(* IEC 61131-3 sources: Mizera_Tube/Plc (part 14) *)

(* ---- RES_IPG.plc ---- *)
*******************************************************************************
*   RES_IPG.PLC
*   ESAutomotion
*   LASER machine
*******************************************************************************
VAR
#include "Cnc.inc"
#include "RemContr.inc"
END_VAR

VAR_IN_OUT
#include "mem.inc"
END_VAR

#include "Iol.inc"
#include "res_ipg.inc"

*******************************************************************************
*   RESONATOR: IPG (YLR / YLS type)
*******************************************************************************
FUNCTION_BLOCK IPG
VAR_INPUT
xSIM:       BOOL;           * Laser in simulation (become from LSR_GEST)
xType:      DWORD;          * 0=YLS, 1=YLR
xReset:     BOOL;           * reset
xEmer:      BOOL;           * emerg
xEmission:  BOOL;           * Emission command
END_VAR

VAR_OUTPUT
yError:     DWORD;          * error
yWarning:   DWORD;          * warning
yState:     BOOL;           * 1=EMISSION ON, 0=EMISSION OFF
END_VAR

VAR
Appoggio:               BOOL;
YLSseries:              BOOL;
YLRseries:              BOOL;
AutoSwitchOn:           BOOL;
Aux_Allarme:            BOOL;
Feedback_Emission_ON:   BOOL;
TON_LASER_REQ:          TON;        * autostart: Laser request OUT
TON_LASER_SWITCH:       TON;        * autostart: Laser switch on OUT
TON_ANALOG_CONTROL:     TON;        * autostart: analog control OUT
TON1:                   TON;        * timeout 1
TON2:                   TON;        * timeout 1
TON3:                   TON;        * timeout 1
RTRIG_RESET:            R_TRIG;     * trigger on reset button
Guide_Las:              BOOL;
CTU_PULS_Guide_Las:     CTU;
RTRIG_REM_GUIDE_LAS:    R_TRIG;
R_TRIG_RemLaserOn:      R_TRIG;
END_VAR

*******************************************************************************
LD   ALWAYS_ZERO                   ** PLCFLAGS.0  Flag sempre stato off
ST   YLSseries
LD   ALWAYS_ONE                    ** PLCFLAGS.1  Flag sempre stato on
ST   YLRseries

LD   xType                         ** 0=YLS, 1=YLR
EQ   0
JMPCN IsYLR

LD   ALWAYS_ONE                    ** PLCFLAGS.1  Flag sempre stato on
ST   YLSseries
LD   ALWAYS_ZERO                   ** PLCFLAGS.0  Flag sempre stato off
ST   YLRseries

IsYLR:

LD   %Par0.0
ANDN (
LD   xReset                        ** reset
ANDN  I_B8_POWER_SUPPLY            ** IPG power supply status
)
ANDN xEmer                         ** emerg
ST   AutoSwitchOn

CAL  TON_LASER_REQ(IN=AutoSwitchOn, PT=0) ** autostart: Laser request OUT

LD   AutoSwitchOn
AND  O_A1_LASER_REQ                ** IPG Richiesta Laser
ST   Appoggio

CAL  TON_LASER_SWITCH(IN=Appoggio, PT=1000) ** autostart: Laser switch on OUT

LD   AutoSwitchOn
AND  O_C1_LASER_SWITCH             ** IPG Laser Switch ON
ST   Appoggio

CAL  TON_ANALOG_CONTROL(IN=Appoggio, PT=1000) ** autostart: analog control OUT

CAL  RTRIG_RESET(CLK=xReset)       ** trigger on reset button

LD   RTRIG_RESET.Q
JMPCN NoReset

LD   0
ST   yError                        ** error
ST   yWarning                      ** warning

LD   ALWAYS_ZERO                   ** PLCFLAGS.0  Flag sempre stato off
ST   yState                        ** 1=EMISSION ON, 0=EMISSION OFF

NoReset:

*******************************************************************************
*   A01 Laser request (wait Laser_ASSIGNED)
*******************************************************************************
CAL  R_TRIG_RemLaserOn(CLK=RemContrLaserOn)
LD   R_TRIG_RemLaserOn.Q
AND  O_A1_LASER_REQ
R    BTN_LASER_REQUEST

LD   R_TRIG_RemLaserOn.Q
ANDN O_A1_LASER_REQ
S    BTN_LASER_REQUEST

LD   BTN_LASER_REQUEST
ANDN AutoSwitchOn
AND  YLSseries
OR (
LD   BTN_LASER_REQUEST
ANDN AutoSwitchOn
AND  YLRseries
AND  I_B8_POWER_SUPPLY             ** IPG power supply status (IW1.6)
)
OR   TON_LASER_REQ.Q
ANDN xSIM                          ** Laser in simulation (become from LSR_GEST)
ST   O_A1_LASER_REQ                ** IPG Richiesta Laser (QW3.11)

*******************************************************************************
*   C01 POWER SUPPLY ON (wait B8 power supply status)
*******************************************************************************
LD   BTN_POWER_ON
ANDN AutoSwitchOn
OR   TON_LASER_SWITCH.Q
AND  O_A1_LASER_REQ                ** IPG Richiesta Laser
AND  I_B7_LASER_ASSIGNED           ** IPG Laser ASSIGNED
ANDN xSIM                          ** Laser in simulation (become from LSR_GEST)
AND  YLSseries
ST   O_C1_LASER_SWITCH             ** IPG Laser Switch ON

*******************************************************************************
*   A05 Guide laser ON
*******************************************************************************
CAL  RTRIG_REM_GUIDE_LAS(CLK:=RemContrGuideLas)        * Xhc_Puls.17 Laser shut

CAL  CTU_PULS_Guide_Las(CU:=RTRIG_REM_GUIDE_LAS.Q,R=CTU_PULS_Guide_Las.Q,PV=2)

LD   CTU_PULS_Guide_Las.CV
EQ   1
ST   Guide_Las

LD   BTN_GUIDE_ON
OR   Guide_Las
ANDN xSIM                          ** Laser in simulation (become from LSR_GEST)
ST   O_A5_GUIDE_LASER              ** IPG Laser spot guide ON

*******************************************************************************
*   A06 Analog control ON
*******************************************************************************
LD   BTN_ANALOG_ON
OR   TON_ANALOG_CONTROL.Q
ANDN xSIM                          ** Laser in simulation (become from LSR_GEST)
ST   O_A6_ANALOG_CONTROL           ** IPG Controllo analogico ON

*******************************************************************************
*   A03 Enable internal control
*******************************************************************************
LD   BTN_INT_ON
ANDN xSIM                          ** Laser in simulation (become from LSR_GEST)
ST   O_A3_INT_CONTROL              ** IPG Abilitazione Controllo interno

*******************************************************************************
*   A04 Reset
*******************************************************************************
LD   BTN_RESET
*OR   xReset                        ** reset
ANDN xSIM                          ** Laser in simulation (become from LSR_GEST)
ST   O_A4_LASER_RESET              ** IPG Resetta errori

*******************************************************************************
*   START PROGRAM
*******************************************************************************
*LD   xEmission                     ** Emission command
*ANDN xSIM                          ** Laser in simulation (become from LSR_GEST)
*ST   O_A2_LASER_PROG_RUN           ** IPG (START PROGRAM)

*******************************************************************************
*   ERROR
*******************************************************************************
*** Allarme errore laser (B4)
LD   I_B4_LASER_ERROR              ** IPG YLS YLR Laser in Alarm status
ST   yError.0

*** Allarme laser non attivo (A2 senza B1)
LD   O_A2_LASER_PROG_RUN           ** IPG (START PROGRAM)
ANDN I_B1_LASER_READY              ** IPG Laser internal main power supply ON (Aux Power ON)
ST   yError.1

*** Allarme laser non assegnato (A1 senza B7)
LD   O_A1_LASER_REQ                ** IPG Richiesta Laser
ANDN I_B7_LASER_ASSIGNED           ** IPG Laser ASSIGNED
ST    Aux_Allarme

CAL  TON1(IN=Aux_Allarme,PT=3000)  ** timeout 1
LD   TON1.Q
ST   yError.2

*** Allarme laser non attivo (C1 senza B8)
LD   O_C1_LASER_SWITCH             ** IPG Laser Switch ON
ANDN I_B8_POWER_SUPPLY             ** IPG power supply status
ST   Aux_Allarme

CAL  TON2(IN=Aux_Allarme,PT=5000)  ** timeout 1
LD   TON2.Q
ST   yError.3

*** Allarme Trascorso tempo massimo attesa segnale emission on dal laser
LD   O_A2_LASER_PROG_RUN           ** IPG (START PROGRAM)
ANDN I_B2_EMISSION_ON              ** IPG Emission ON
ST   Feedback_Emission_ON

CAL  TON3(IN=Feedback_Emission_ON,PT=3000) ** timeout 1

LD   TON3.Q
ST   yError.4

*******************************************************************************
*   WARNING
*******************************************************************************
*** Messaggio laser in stato di pre-allarme (B13)

LD   I_B13_AVVERTENZA              ** IPG WARNING OUT
ST   yWarning.0

LD   O_A2_LASER_PROG_RUN           ** IPG (START PROGRAM)
***AND  I_B2_EMISSION_ON              ** IPG Emission ON
ST   yState                        ** 1=EMISSION ON, 0=EMISSION OFF

*******************************************************************************
*   HMI
*******************************************************************************

*** Buttons

LD   O_A1_LASER_REQ                ** IPG Richiesta Laser
ST   %Leds0.0
LD   O_C1_LASER_SWITCH             ** IPG Laser Switch ON
ST   %Leds0.1
LD   O_A4_LASER_RESET              ** IPG Resetta errori
ST   %Leds0.2
LD   O_A3_INT_CONTROL              ** IPG Abilitazione Controllo interno
ST   %Leds0.3
LD   O_A6_ANALOG_CONTROL           ** IPG Controllo analogico ON
ST   %Leds0.4
LD   O_A5_GUIDE_LASER              ** IPG Laser spot guide ON
ST   %Leds0.5
LD   O_A2_LASER_PROG_RUN           ** IPG (START PROGRAM)
ST   %Leds0.6

*** Feedback

LD   I_B7_LASER_ASSIGNED           ** IPG Laser ASSIGNED
ST   %Leds1.0
LD   I_B8_POWER_SUPPLY             ** IPG power supply status
ST   %Leds1.1
LD   I_B3_INT_CONTROL              ** IPG Controllo interno abilitato
ST   %Leds1.2
LD   I_B6_ANALOG_CONTROL           ** IPG Controllo analogico ON
ST   %Leds1.3
LD   I_B5_LASER_GUIDE              ** IPG Laser guida ON
ST   %Leds1.4
LD   I_B1_LASER_READY              ** IPG Laser internal main power supply ON (Aux Power ON)
ST   %Leds1.5
LD   I_B2_EMISSION_ON              ** IPG Emission ON
ST   %Leds1.6
LD   I_B13_AVVERTENZA              ** IPG WARNING OUT
ST   %Leds1.7
LD   I_B4_LASER_ERROR              ** IPG YLS YLR Laser in Alarm status
ST   %Leds1.8

*** If laser in simulation

LD   xSIM                          ** Laser in simulation (become from LSR_GEST)
JMPCN NoLaserInSIM
LD   0
ST   yError                        ** error
ST   yWarning                      ** warning

LD   xEmission                     ** Emission command
ST   yState                        ** 1=EMISSION ON, 0=EMISSION OFF
NoLaserInSIM:

END_FUNCTION_BLOCK

(* ---- RestFB.plc ---- *)
**************************************************
* New state machine to restart the machine after
* an hold command or tip touch event
**************************************************

FUNCTION_BLOCK Restart_Cut

VAR
State:              DWORD;
ActualAttempts:     DWORD;
PrevCountAttempt:   DWORD;
RetraceTimeout:     DWORD;

ResetCounter:       BOOL;
MaxAttemptsDone:    BOOL;

TON_RETR_DONE:      TON;
TON_RESCOUNT:       TON;
FTRIG_END_RETRACE:  F_TRIG;

END_VAR

VAR_INPUT
xProg_Run:      BOOL;
xTip_Touch:     BOOL;
xZupExecuted:   BOOL;
xMachineInHold: BOOL;
xRetraceOn:     BOOL;
xAttempts:      DWORD;
END_VAR

VAR_OUTPUT
yZupRequest:    BOOL;
yStartRetrace:  BOOL;
yStartProg:     BOOL;
yHoldProg:      BOOL;
yInibTipTouch:  BOOL;
END_VAR

*********************************************************************

LD   3000
ST   RetraceTimeout

LDN  xProg_Run
JMPCN no_ResetVar

LD   0
ST   yZupRequest
ST   yStartRetrace
ST   yStartProg
ST   yHoldProg
ST   yInibTipTouch
ST   State

LD   1
ST   ActualAttempts
ST   PrevCountAttempt
no_ResetVar:

*****************************
* Attempt counter

LD   ActualAttempts
GT   xAttempts
ST   MaxAttemptsDone

LD   ActualAttempts
EQ   PrevCountAttempt
ANDN MaxAttemptsDone
ST   ResetCounter

CAL  TON_RESCOUNT (IN:=ResetCounter,PT:=20000)

LD   TON_RESCOUNT.Q
JMPCN no_res_count
LD   0
ST   PrevCountAttempt
ST   ActualAttempts
no_res_count:
******************************

*********************************************************************
*   STATO=0
*   In case of tip touch this state makes a request to the regulator
*   to bring up the head
*********************************************************************
LD   State
EQ   0
JMPCN STATE0_end

R    yStartProg

LD   ActualAttempts
ST   PrevCountAttempt

LD   xTip_Touch
AND  xProg_Run
ANDN MaxAttemptsDone
JMPCN STATE0_endif_A

** assume stay here just one scan
LD  ActualAttempts
ADD 1
ST  ActualAttempts
**

S   yZupRequest
S   yInibTipTouch

LD  10
ST  State

STATE0_endif_A:
JMP state_machine_end

STATE0_end:

CAL  TON_RETR_DONE (IN:=yStartRetrace,PT:=RetraceTimeout)
CAL  FTRIG_END_RETRACE(CLK=xRetraceOn)

*********************************************************************
*   STATO=10
*   Wait that the machine is in hold then send the request of retrace back
*********************************************************************
LD   State
EQ   10
JMPCN STATE10_end

LD   xZupExecuted
AND  xMachineInHold
JMPCN STATE10_endif_A

S  yStartRetrace

LD  11
ST  State

STATE10_endif_A:
JMP state_machine_end

STATE10_end:

*********************************************************************
*   STATO=11
*   Wait that the machine is in hold then send the request of retrace back
*********************************************************************
LD   State
EQ   11
JMPCN STATE11_end

LD   FTRIG_END_RETRACE.Q
OR (
LD   TON_RETR_DONE.Q
ANDN xRetraceOn
)
JMPCN no_retrace_end

R   yStartRetrace
R   yInibTipTouch
R   yZupRequest
S   yStartProg

LD  0
ST  State

no_retrace_end:
JMP state_machine_end

STATE11_end:

*********************************************************************
state_machine_end:

END_FUNCTION_BLOCK

(* ---- RToolSur.plc ---- *)
*=========================================================================
* VRTC GATEWAY VARIABLES SECTION
*=========================================================================
#funcdec "ASSI.plc"
#funcdec "CNC.plc"
#funcdec "StatMReg.plc"

VAR
REG_MAC:  REG_STATE_MACHINE;
vrtcExTool:         VRTC_EX;
vrtcExSurface:      VRTC_EX;

plcVrtcHandling:       BOOL;
firstCallToPlcHandler:  BOOL;

toolCommandToggle:      BOOL;
surfaceCommandToggle:   BOOL;
appoggio:               BOOL;

TR_ToolVrtcToggle:      TRIG;
TR_SurfaceVrtcToggle:   TRIG;
RTR_PlcVrtcHandling:    R_TRIG;
cosAngle:               DWORD;
ActVPBSelect:           DWORD;
TP_reset:               TP;

SensorGain:             DWORD;

END_VAR

VAR_IN_OUT
UVH_COMMAND_0                          AT %uvhCommand0;
UVH_COMMAND_MACHINE_MODE               AT %uvhCommand1;
UVH_COMMAND_PLC_VRTC_HANDLING          AT %uvhCommand0.1;
UVH_COMMAND_START_COMMAND              AT %uvhCommand0.2;
UVH_COMMAND_FREEZE_REGOL               AT %uvhCommand0.3;
UVH_COMMAND_JUMP                       AT %uvhCommand0.4;
UVH_COMMAND_L10                        AT %uvhCommand0.5;
UVH_COMMAND_L3                         AT %uvhCommand0.6;
UVH_STATUS_PLC_VRTC_HANDLING           AT %uvhStatus0.1;
UVH_STATUS_MACHINE_MODE                AT %uvhStatus1;
UVH_STATUS_COMMAND_RUNNING             AT %uvhStatus0.2;

UVH_TOOL_COMMAND_RESET                 AT %uvhToolCommand0.0;
UVH_TOOL_COMMAND_SIMUL                 AT %uvhToolCommand0.1;
UVH_TOOL_COMMAND_MOVE_TO_TARGET        AT %uvhToolCommand0.2;
UVH_TOOL_COMMAND_RES_POS_INT           AT %uvhToolCommand0.3;
UVH_TOOL_COMMAND_POS_LIM_DISAB         AT %uvhToolCommand0.4;
UVH_TOOL_COMMAND_DE_OVERLAP_ENAB       AT %uvhToolCommand0.5;
UVH_TOOL_COMMAND_ERROR_AMP_ENAB        AT %uvhToolCommand0.6;
UVH_TOOL_COMMAND_TOGGLE                AT %uvhToolCommand0.31;
UVH_TOOL_COMMAND_SIM_OFFSET_SET        AT %uvhToolCommand1;
UVH_TOOL_COMMAND_SETPOINT              AT %uvhToolCommand2;
UVH_TOOL_COMMAND_VECTOR_SELECT         AT %uvhToolCommand3;

UVH_TOOL_STATUS_SIGNAL_LOCK            AT %uvhToolStatus0.2;
UVH_TOOL_STATUS_TOGGLE_ACK             AT %uvhToolStatus0.31;
UVH_TOOL_STATUS_SIM_OFFSET_CUR         AT %uvhToolStatus1;
UVH_TOOL_STATUS_FLT_Q                  AT %uvhToolStatus2;

UVH_SURFACE_COMMAND_RESET              AT %uvhSurfaceCommand0.0;
UVH_SURFACE_COMMAND_SIMUL              AT %uvhSurfaceCommand0.1;
UVH_SURFACE_COMMAND_MOVE_TO_TARGET     AT %uvhSurfaceCommand0.2;
UVH_SURFACE_COMMAND_RES_POS_INT        AT %uvhSurfaceCommand0.3;
UVH_SURFACE_COMMAND_POS_LIM_DISAB      AT %uvhSurfaceCommand0.4;
UVH_SURFACE_COMMAND_DE_OVERLAP_ENAB    AT %uvhSurfaceCommand0.5;
UVH_SURFACE_COMMAND_ERROR_AMP_ENAB     AT %uvhSurfaceCommand0.6;
UVH_SURFACE_COMMAND_TOGGLE             AT %uvhSurfaceCommand0.31;
UVH_SURFACE_COMMAND_SIM_OFFSET_SET     AT %uvhSurfaceCommand1;
UVH_SURFACE_COMMAND_SETPOINT           AT %uvhSurfaceCommand2;
UVH_SURFACE_COMMAND_VECTOR_SELECT      AT %uvhSurfaceCommand3;

UVH_SURFACE_STATUS_SIGNAL_LOCK         AT %uvhSurfaceStatus0.2;
UVH_SURFACE_STATUS_TOGGLE_ACK          AT %uvhSurfaceStatus0.31;
UVH_SURFACE_STATUS_SIM_OFFSET_CUR      AT %uvhSurfaceStatus1;
UVH_SURFACE_STATUS_FLT_Q               AT %uvhSurfaceStatus2;

VRMON_Q_FLT_Q                          AT %VrMon_Q_Flt_Q;
VrSensorGain                          AT %VrSensorGain;
END_VAR

FUNCTION_BLOCK REG_T_S

VAR_INPUT

* Tool VRTC Input

xToolVrtcSetPoint:       DWORD;
xToolVrtcId:            DWORD;
xToolSim:                BOOL;

xLimDownSpeed:            BOOL;

xSensorRes:              DWORD;         * Capacitive sensor resolution (4095,32767,65535)
xNextPos_X_Jump_VRTC:    DWORD;         * X setpoint coordinate for jump
xNextPos_Y_Jump_VRTC:    DWORD;         * Y setpoint coordinate for jump
xNextPos_C_Jump_VRTC:    DWORD;         * C setpoint coordinate for jump
xNextPos_Z_Jump_VRTC:    DWORD;         * Z setpoint coordinate for jump

xInit_X_Posit_VRTC:      DWORD;         * X init jump position
xInit_Y_Posit_VRTC:      DWORD;         * Y init jump position
xInit_C_Posit_VRTC:      DWORD;         * C init jump position
xInit_Z_Posit_VRTC:      DWORD;         * C init jump position

xNextSetpVRTC:           DWORD;         * Setpoint after jump
xPrevSetpVRTC:           DWORD;         * last setpoint before jump
xDistEnabRegulVRTC:      DWORD;         * Distance from target to enab regulation during jump
xZDistStopProbeJVRTC:    DWORD;         * distance along Z to disable the probe vpbselector during jump

xActual_X_Posit_VRTC:    DWORD;         * X Actual position
xActual_Y_Posit_VRTC:    DWORD;         * Y Actual position
xActual_C_Posit_VRTC:    DWORD;         * C Actual position
xActual_Z_Posit_VRTC:    DWORD;         * Z Actual position

* Surface VRTC Input

xSurfVrtcId:            DWORD;
xSurfaceSim:            BOOL;
xLimSpeedPierc:           BOOL;
xAngleBev:              DWORD;
xSpeedForPiercing:        DWORD;                 * Speed for Z axi during piercing

xHead:                  DWORD;
xChannel:               DWORD;
xZtcp:                  DWORD;
xProbThreshold:         DWORD;
xSensorRange:           DWORD;
xFirstFirCost_VRTC:     DWORD;         * ms
xSecondFirCost_VRTC:    DWORD;         * ms
xDelayCost_VRTC:        DWORD;         * ms
xMove_Z_SetP_VRTC:        DWORD;

xMove_Z_VRTC:           BOOL;
xHold_VRTC:             BOOL;
xRealTimeFreeze:         BOOL;

END_VAR

VAR_OUTPUT
yWaitVRTC:               BOOL;
yIncSetPReachedVRTC:     BOOL;
yL3SetpointReachedVRTC:   BOOL;
END_VAR
*=========================================================================
* VRTC GATEWAY SECTION
*=========================================================================
***
* Vrtc Sensor gain settings

LD   xSensorRes
MUL  10000
DIV  xSensorRange
MUL  100
ST   SensorGain

PATH    %vrtc[xToolVrtcId]
LD   SensorGain
ST   VrSensorGain

PATH    %vrtc[xSurfVrtcId]
LD   SensorGain
ST   VrSensorGain

**

*** COMMON ***

LDN     %rc8.21                     * M_IDLE
JMPC    skip_vrtc_idle

    LD      0
    ST      UVH_COMMAND_0

skip_vrtc_idle:

LD      UVH_COMMAND_PLC_VRTC_HANDLING
ST      plcVrtcHandling

*** TOOL VRTC ***

* in cima
LD      UVH_TOOL_COMMAND_TOGGLE
ST      toolCommandToggle

CAL     TR_ToolVrtcToggle(CLK=toolCommandToggle)
LDN     TR_ToolVrtcToggle.Q
JMPC    skip_tool_vrtc_uvh_control

LD      UVH_TOOL_COMMAND_VECTOR_SELECT
ST      vrtcExTool.xVectorSelect

LD      UVH_TOOL_COMMAND_RESET
ST      vrtcExTool.xReset

LD      UVH_TOOL_COMMAND_SIMUL
ST      vrtcExTool.xSimul

LD      UVH_TOOL_COMMAND_MOVE_TO_TARGET
ST      vrtcExTool.xMoveToTarget

LD      UVH_TOOL_COMMAND_RES_POS_INT
ST      vrtcExTool.xResPosInt

LD      UVH_TOOL_COMMAND_POS_LIM_DISAB
ST      vrtcExTool.xPosLimDisab

LD      UVH_TOOL_COMMAND_DE_OVERLAP_ENAB
ST      vrtcExTool.xDeOverlapEnab

LD      UVH_TOOL_COMMAND_ERROR_AMP_ENAB
ST      vrtcExTool.xErrorAmpEnab

LD      UVH_TOOL_COMMAND_SIM_OFFSET_SET
ST      vrtcExTool.xSimOffsetSet

LD      UVH_TOOL_COMMAND_SETPOINT
ST      vrtcExTool.xSetPoint

skip_tool_vrtc_uvh_control:

*** SURFACE VRTC ***

* in cima
LD      UVH_SURFACE_COMMAND_TOGGLE
ST      surfaceCommandToggle

CAL     TR_SurfaceVrtcToggle(CLK=surfaceCommandToggle)
LDN     TR_SurfaceVrtcToggle.Q
JMPC    skip_surface_vrtc_uvh_control

LD      UVH_SURFACE_COMMAND_VECTOR_SELECT
ST      vrtcExSurface.xVectorSelect

LD      UVH_SURFACE_COMMAND_RESET
ST      vrtcExSurface.xReset

LD      UVH_SURFACE_COMMAND_SIMUL
ST      vrtcExSurface.xSimul

LD      UVH_SURFACE_COMMAND_MOVE_TO_TARGET
ST      vrtcExSurface.xMoveToTarget

LD      UVH_SURFACE_COMMAND_RES_POS_INT
ST      vrtcExSurface.xResPosInt

LD      UVH_SURFACE_COMMAND_POS_LIM_DISAB
ST      vrtcExSurface.xPosLimDisab

LD      UVH_SURFACE_COMMAND_DE_OVERLAP_ENAB
ST      vrtcExSurface.xDeOverlapEnab

LD      UVH_SURFACE_COMMAND_ERROR_AMP_ENAB
ST      vrtcExSurface.xErrorAmpEnab

LD      UVH_SURFACE_COMMAND_SIM_OFFSET_SET
ST      vrtcExSurface.xSimOffsetSet

LD      UVH_SURFACE_COMMAND_SETPOINT
ST      vrtcExSurface.xSetPoint

skip_surface_vrtc_uvh_control:

LDN     plcVrtcHandling
JMPCN   reset_vbselect

LD      0
ST      %vpbSelectors0

reset_vbselect:

*** COMMON ***

CAL     RTR_PlcVrtcHandling(CLK=plcVrtcHandling)
LD      RTR_PlcVrtcHandling.Q
ST      firstCallToPlcHandler

LDN     plcVrtcHandling
JMPC    skip_plc_handling
*XXX DO YOUR OWN PLC HANDLING cambio setpoint etc

 LD      xAngleBev                   * Bevel angle ofthe head
 COS
 ST      cosAngle

* State Machine FB

 LD      vrtcExSurface.xSimul
 ST      REG_MAC.xISO_S_SimEnab

 LD      vrtcExSurface.xErrorAmpEnab
 ST      REG_MAC.xISO_S_ErrAmp

 LD      vrtcExTool.xSimul
 ST      REG_MAC.xISO_T_SimEnab

 LD      vrtcExTool.xSetPoint
 ST      REG_MAC.xISO_T_SetPoint

 LD      vrtcExTool.xErrorAmpEnab
 ST      REG_MAC.xISO_T_ErrAmp

 LD      xFirstFirCost_VRTC
 ST      REG_MAC.xFirstFirCost         * ms

 LD      xSecondFirCost_VRTC
 ST      REG_MAC.xSecondFirCost        * ms

 LD      xDelayCost_VRTC
 ST      REG_MAC.xDelayCost         * ms

 LD      firstCallToPlcHandler
 ST      REG_MAC.xFirstPlcHandling

 LD      xProbThreshold
 ST      REG_MAC.xProbThres

 LD      xZtcp
 ST      REG_MAC.xZ_TCP

 LD      UVH_COMMAND_MACHINE_MODE
 ST      REG_MAC.xIsoPhase

 LD      vrtcExTool.yBusy
 ST      REG_MAC.xToolBusy

 LD      vrtcExSurface.yBusy
 ST      REG_MAC.xSurfaceBusy

 LD      vrtcExTool.ySignalLock
 ST      REG_MAC.xToolSignalLock

 LD      vrtcExSurface.ySignalLock
 ST      REG_MAC.xSurfSignalLock

 LD      xToolVrtcSetPoint         * [um]
 DIV     10
 ST      REG_MAC.xSetpoint

 LD      UVH_COMMAND_START_COMMAND
 ST      REG_MAC.xStartEx

 LD      xSensorRange
 ST      REG_MAC.xSensorRange

 LD      UVH_COMMAND_FREEZE_REGOL
 OR      xRealTimeFreeze
 ST      REG_MAC.xFreezeRegol

 LD      xNextPos_Y_Jump_VRTC          * Y setpoint coordinate for jump
 ST      REG_MAC.xNextPos_Y_Jump

 LD      xNextPos_X_Jump_VRTC          * X setpoint coordinate for jump
 ST      REG_MAC.xNextPos_X_Jump

 LD      xNextPos_C_Jump_VRTC          * C setpoint coordinate for jump
 ST      REG_MAC.xNextPos_C_Jump

 LD      xNextPos_Z_Jump_VRTC          * Z setpoint coordinate for jump
 ST      REG_MAC.xNextPos_Z_Jump

 LD      xInit_Y_Posit_VRTC            * Y init jump position
 ST      REG_MAC.xInit_Y_Posit

 LD      xInit_X_Posit_VRTC            * X init jump position
 ST      REG_MAC.xInit_X_Posit

 LD      xInit_C_Posit_VRTC            * C init jump position
 ST      REG_MAC.xInit_C_Posit

 LD      xInit_Z_Posit_VRTC            * Z init jump position
 ST      REG_MAC.xInit_Z_Posit

 LD      xActual_X_Posit_VRTC          * X Actual position
 ST      REG_MAC.xActual_X_Posit

 LD      xActual_C_Posit_VRTC          * C Actual position
 ST      REG_MAC.xActual_C_Posit

 LD      xActual_Z_Posit_VRTC          * C Actual position
 ST      REG_MAC.xActual_Z_Posit

 LD      xActual_Y_Posit_VRTC          * Y Actual position
 ST      REG_MAC.xActual_Y_Posit

 LD      UVH_COMMAND_JUMP
 ST      REG_MAC.xJumpReq

 LD      UVH_COMMAND_L3
 ST      REG_MAC.xJumpL3Req

 LD      xNextSetpVRTC
 ST      REG_MAC.xNextSetp

 LD      xPrevSetpVRTC
 ST      REG_MAC.xPrevSetp

 LD      xDistEnabRegulVRTC
 ST      REG_MAC.xDistEnabRegul

 LD      UVH_COMMAND_L10
 ST      REG_MAC.xL10Req

*
 LD      xZDistStopProbeJVRTC
 ST      REG_MAC.xZDistStopProbeJ

 LD      cosAngle
 ST      REG_MAC.xCosBevelAngle

PATH    %vrtc[xToolVrtcId]

 LD      VRMON_Q_FLT_Q
 ST      REG_MAC.xToolFlt_Q

* Hold and move head up during cutting

 LD      xMove_Z_VRTC
 ST      REG_MAC.xMove_Z

 LD      xMove_Z_SetP_VRTC
 DIV     10
 ST      REG_MAC.xMove_Z_SetP

* Hold

 LD      xHold_VRTC
 ST      REG_MAC.xHold

 CAL     REG_MAC

 * Hand-shake signals

 LD      REG_MAC.yStateMachinePhase
 ST      UVH_STATUS_MACHINE_MODE

 LD      REG_MAC.yComRunning
 ST      UVH_STATUS_COMMAND_RUNNING

 LD      REG_MAC.yVPBSelect
 ST      ActVPBSelect
 ST      %vpbSelectors0

 LD      REG_MAC.yWait
 ST      yWaitVRTC

 LD      REG_MAC.yIncSetPReached
 ST      yIncSetPReachedVRTC

 LD      REG_MAC.yL3SetpointReached
 ST      yL3SetpointReachedVRTC

 * Tool Vrtc plc handling

 LD      REG_MAC.y_T_SimEnab
 ST      vrtcExTool.xSimul

 LD      REG_MAC.y_T_SetPoint
 ST      vrtcExTool.xSetPoint

 LD      REG_MAC.y_T_ErrAmp
 ST      vrtcExTool.xErrorAmpEnab

 * Surface Vrtc plc handling

 LD      REG_MAC.y_S_SimEnab
 ST      vrtcExSurface.xSimul

 LD      REG_MAC.y_S_SetPoint
 ST      vrtcExSurface.xSetPoint

 LD      REG_MAC.y_S_ErrAmp
 ST      vrtcExSurface.xErrorAmpEnab

skip_plc_handling:

*XXX DO YOUR OWN PLC RESET LOGIC

LDN     %rc8.0
JMPCN no_reset

LD      0
ST      vrtcExTool.xErrorAmpEnab
ST      vrtcExSurface.xErrorAmpEnab
ST      UVH_STATUS_MACHINE_MODE
ST      ActVPBSelect
ST      UVH_STATUS_MACHINE_MODE
ST      UVH_STATUS_COMMAND_RUNNING
ST      UVH_COMMAND_FREEZE_REGOL
ST      UVH_COMMAND_JUMP
ST      UVH_COMMAND_L3
ST      UVH_COMMAND_L10
ST      yWaitVRTC
ST      yIncSetPReachedVRTC

LD      1
ST      vrtcExTool.xReset           * Reset
ST      vrtcExSurface.xReset        * Reset
ST      vrtcExTool.xSimul
ST      vrtcExSurface.xSimul

no_reset:

LD      ActVPBSelect
EQ      0
JMPCN   end_selector0
*// 0) INITIAL PROBING
PATH    %vpbs0
end_selector0:

LD      ActVPBSelect
EQ      1
JMPCN   end_selector1
*// 1) JUMP parameters
PATH    %vpbs1
end_selector1:

LD      ActVPBSelect
EQ      2
JMPCN   end_selector2
*// 2) FAR parameters (jump to pierce/probing point, etc)
PATH    %vpbs2
end_selector2:

LD      ActVPBSelect
EQ      3
JMPCN   end_selector3
*// 3) NEAR parameters (probing to piercing, piercing to cutting point, etc)
PATH    %vpbs3
end_selector3:

LD      ActVPBSelect
EQ      4
JMPCN   end_selector4
*// 4) CUT parameters
PATH    %vpbs4
end_selector4:

LD      ActVPBSelect
EQ      5
JMPCN   end_selector5
*// 5) Hold parameters
PATH    %vpbs5
end_selector5:

LD      ActVPBSelect
EQ      6
JMPCN   end_selector6
*// 6) Simulation parameters
PATH    %vpbs6
end_selector6:

*** TOOL VRTC ***

LD      %PLCFLAGS.1
ST      vrtcExTool.xMLonlyClampFilterIn
ST      vrtcExTool.xMLonlyClampFilterInDot

*//XXX replace with table parameters
LD      %vpbp0
ST      vrtcExTool.xUpPosLimit

LD      %vpbp1
ST      vrtcExTool.xLwPosLimit

* Capacitive test in progress
LD      %C18.17
JMPCN   NOLWPOSLIMT
LD      -9999999
ST      vrtcExTool.xLwPosLimit
NOLWPOSLIMT:

LD      %vpbp2
ST      vrtcExTool.xVelLimitUp

LD      %vpbp3
ST      vrtcExTool.xVelLimitDown

LD      %vpbp4
ST      vrtcExTool.xAccLimitUp

LD      %vpbp5
ST      vrtcExTool.xAccLimitDown

LD      %vpbp6
ST      vrtcExTool.xKpGain

LD      %vpbp7
ST      vrtcExTool.xKpTransPtr

LD      %vpbp8
ST      vrtcExTool.xKpTransMul

LD      %vpbp9
ST      vrtcExTool.xDbPos

LD      %vpbp10
ST      vrtcExTool.xDbNeg

LD      %vpbp11
ST      vrtcExTool.xFilterCutOff

LD      %vpbp12
ST      vrtcExTool.xFilterDamping

LD      %vpbp13
ST      vrtcExTool.xSimFadingTime

LD      %vpbp14
ST      vrtcExTool.xLockVelLimitUp

LD      %vpbp15
ST      vrtcExTool.xLockVelLimitDown

LD      xLimSpeedPierc
JMPCN   no_lim_speed1
 LD      xSpeedForPiercing                  * Speed for Z axi during piercing
 ST      vrtcExTool.xVelLimitDown
 ST      vrtcExTool.xVelLimitUp

LD      5
ST      vrtcExTool.xLockVelLimitUp
ST      vrtcExTool.xLockVelLimitDown

no_lim_speed1:

LD      %vpbp17
ST      vrtcExTool.xSlidingDecel

LD      %vpbp16
ST      vrtcExTool.xLockAccLimit
*//XXX replace with table parameters
PATH    %vrtc[xToolVrtcId]
CAL     vrtcExTool

LD      vrtcExTool.ySignalLock
ST      UVH_TOOL_STATUS_SIGNAL_LOCK

LD      vrtcExTool.ySimOffsetCur
ST      UVH_TOOL_STATUS_SIM_OFFSET_CUR

LD      vrtcExTool.yFltQ
ST      UVH_TOOL_STATUS_FLT_Q

* in fondo
LD      vrtcExTool.yBusy
JMPC    skip_tool_toggle_update

    LD      toolCommandToggle
    ST      UVH_TOOL_STATUS_TOGGLE_ACK

skip_tool_toggle_update:

*** SURFACE VRTC ***

LD      %PLCFLAGS.1
ST      vrtcExSurface.xMLonlyClampFilterIn
ST      vrtcExSurface.xMLonlyClampFilterInDot

*//XXX replace with table parameters
LD      %vpbp0
ST      vrtcExSurface.xUpPosLimit

LD      %vpbp1
ST      vrtcExSurface.xLwPosLimit

* Capacitive test in progress
LD      %C18.17
JMPCN   NOLWPOSLIMS
LD      -9999999
ST      vrtcExSurface.xLwPosLimit
NOLWPOSLIMS:

LD      %vpbp2
ST      vrtcExSurface.xVelLimitUp

LD      xLimDownSpeed
JMPCN   no_0_speed
        LD      1
        ST      vrtcExSurface.xVelLimitDown
JMP no_0_com
no_0_speed:
        LD      %vpbp3
        ST      vrtcExSurface.xVelLimitDown
no_0_com:

LD      %vpbp4
ST      vrtcExSurface.xAccLimitUp

LD      %vpbp5
ST      vrtcExSurface.xAccLimitDown

LD      %vpbp6
ST      vrtcExSurface.xKpGain

LD      %vpbp7
ST      vrtcExSurface.xKpTransPtr

LD      %vpbp8
ST      vrtcExSurface.xKpTransMul

LD      %vpbp9
ST      vrtcExSurface.xDbPos

LD      %vpbp10
ST      vrtcExSurface.xDbNeg

LD      %vpbp11
ST      vrtcExSurface.xFilterCutOff

LD      %vpbp12
ST      vrtcExSurface.xFilterDamping

LD      %vpbp13
ST      vrtcExSurface.xSimFadingTime

LD      %vpbp14
ST      vrtcExSurface.xLockVelLimitUp

LD      %vpbp15
ST      vrtcExSurface.xLockVelLimitDown

LD      xLimSpeedPierc
JMPCN   no_lim_speed
 LD      xSpeedForPiercing                  * Speed for Z axi during piercing
 ST      vrtcExSurface.xVelLimitDown
 ST      vrtcExSurface.xVelLimitUp

 LD      5
 ST      vrtcExSurface.xLockVelLimitUp
 ST      vrtcExSurface.xLockVelLimitDown

no_lim_speed:

LD      %vpbp16
ST      vrtcExSurface.xLockAccLimit

LD      %vpbp17
ST      vrtcExSurface.xSlidingDecel

*//XXX replace with table parameters
PATH    %vrtc[xSurfVrtcId]
CAL     vrtcExSurface

LD      vrtcExSurface.ySignalLock
ST      UVH_SURFACE_STATUS_SIGNAL_LOCK

LD      vrtcExSurface.ySimOffsetCur
ST      UVH_SURFACE_STATUS_SIM_OFFSET_CUR

LD      vrtcExSurface.yFltQ
ST      UVH_SURFACE_STATUS_FLT_Q

* in fondo
LD      vrtcExSurface.yBusy
JMPC    skip_surface_toggle_update

    LD      surfaceCommandToggle
    ST      UVH_SURFACE_STATUS_TOGGLE_ACK

skip_surface_toggle_update:

*** COMMON ***

LD      vrtcExTool.yBusy
OR      vrtcExSurface.yBusy
JMPC    skip_vrtc_handling_state_update

    LD      plcVrtcHandling
    ST      UVH_STATUS_PLC_VRTC_HANDLING
skip_vrtc_handling_state_update:

END_FUNCTION_BLOCK

(* ---- SetVasca.plc ---- *)
**************************************************************************
*   SETVASCA.PLC
**************************************************************************
#funcdec "assi.plc"
#funcdec "mand.plc"
#funcdec "cnc.plc"

VAR
#include "assi.inc"
#include "cnc.inc"
END_VAR

#include "iol.inc"

**************************************************************************
* FB GESTVS
**************************************************************************
FUNCTION_BLOCK GESTVS

VAR_INPUT
xStartX:        DWORD;  * Quota X0 inizio vasca (micron)
xEndX:          DWORD;  * Quota X1 fine vasca (micron)
xStartY:        DWORD;  * Quota Y0 inizio vasca (micron)
xEndY:          DWORD;  * Quota Y1 fine vasca (micron)
END_VAR

VAR_OUTPUT
yVascaOn:       BOOL;   * Apri vasca
END_VAR

VAR
locX:           DWORD;
locY:           DWORD;
XactualQta:     DWORD;  * X actual quota
YactualQta:     DWORD;  * Y actual quota
MinLimit:       DWORD;  * Minimum Limit
MaxLimit:       DWORD;  * Maximum Limit
insideLimitX:   BOOL;   *
insideLimitY:   BOOL;   *
appoggio:       BOOL;   * Apri vasca
TOF_VASC:       TOF;
END_VAR

****************************************
*   Find the X and Y head coordinate
****************************************
LD   %GenVasche.GV_ParB0    ** 5 axes machine
JMPCN Normal

PATH %ax[%GenVasche.GV_ParB1]

LD   %ra54              ** X TCP
ST   locX

PATH %ax[%GenVasche.GV_ParB2]

LD   %ra54              ** Y TCP
ST   locY

LD   %cn0.mat.sts0
EQ   16#B
JMPCN identity

LD   locX
DIV  100                ** DIV per problemi di overflow
MUL  %cn0.mat.a0
ADD  (
LD   locY
DIV  100                ** DIV per problemi di overflow
MUL  %cn0.mat.a1
)
DIV  10
ADD  (
LD   %cn0.mat.a3
DIV  1000
)
ST   XactualQta                    ** X actual quota

LD   locX
DIV  100                ** DIV per problemi di overflow
MUL  %cn0.mat.a4
ADD  (
LD   locY
DIV  100                ** DIV per problemi di overflow
MUL  %cn0.mat.a5
)
DIV  10
ADD  (
LD   %cn0.mat.a7
DIV  1000
)
ST   YactualQta                    ** Y actual quota

JMP  ComHead

identity:
LD   locX
ST   XactualQta                    ** X actual quota

LD   locY
ST   YactualQta                    ** Y actual quota

JMP  ComHead

Normal:
PATH %ax[%GenVasche.GV_ParB1]
LD   %ra4
ST   XactualQta                    ** X actual quota

PATH %ax[%GenVasche.GV_ParB2]
LD   %ra4
ST   YactualQta                    ** Y actual quota

ComHead:
****************************************
*   Check with X axis
****************************************
LD   xStartX                       ** Quota X0 inizio vasca (micron)
SUB  %GenVasche.GV_ParDW0   * Sovrapposizione
ST   MinLimit                      ** Minimum Limit

LD   xEndX                         ** Quota X1 fine vasca (micron)
ADD  %GenVasche.GV_ParDW0   * Sovrapposizione
ST   MaxLimit                      ** Maximum Limit

LD   XactualQta                    ** X actual quota
GT   MinLimit                      ** Minimum Limit
AND(
LD   XactualQta                    ** X actual quota
LT   MaxLimit                      ** Maximum Limit
)
ST   insideLimitX                  **

****************************************
*   Check with Y axis
****************************************
LD   xStartY                       ** Quota Y0 inizio vasca (micron)
SUB  %GenVasche.GV_ParDW0   * Sovrapposizione
ST   MinLimit                      ** Minimum Limit

LD   xEndY                         ** Quota Y1 fine vasca (micron)
ADD  %GenVasche.GV_ParDW0   * Sovrapposizione
ST   MaxLimit                      ** Maximum Limit

LD   YactualQta                    ** Y actual quota
GT   MinLimit                      ** Minimum Limit
AND(
LD   YactualQta                    ** Y actual quota
LT   MaxLimit                      ** Maximum Limit
)
ST   insideLimitY                  **

****************************************
*   Check if open or not
****************************************
LD   insideLimitX                  **
AND  insideLimitY                  **
ST   appoggio                      ** Apri vasca

CAL  TOF_VASC(IN=appoggio, PT=%GenVasche.GV_ParDW1) ** Apri vasca

LD   TOF_VASC.Q
ST   yVascaOn                      ** Apri vasca

END_FUNCTION_BLOCK

**************************************************************************

VAR

VASCA0:         GESTVS;
VASCA1:         GESTVS;
VASCA2:         GESTVS;
VASCA3:         GESTVS;
VASCA4:         GESTVS;
VASCA5:         GESTVS;
VASCA6:         GESTVS;
VASCA7:         GESTVS;
VASCA8:         GESTVS;
VASCA9:         GESTVS;
VASCA10:        GESTVS;
VASCA11:        GESTVS;
VASCA12:        GESTVS;
VASCA13:        GESTVS;
VASCA14:        GESTVS;
VASCA15:        GESTVS;
VASCA16:        GESTVS;
VASCA17:        GESTVS;
VASCA18:        GESTVS;
VASCA19:        GESTVS;
VASCA20:        GESTVS;
VASCA21:        GESTVS;
VASCA22:        GESTVS;
VASCA23:        GESTVS;
VASCA24:        GESTVS;
VASCA25:        GESTVS;
VASCA26:        GESTVS;
VASCA27:        GESTVS;
VASCA28:        GESTVS;
VASCA29:        GESTVS;
VASCA30:        GESTVS;
VASCA31:        GESTVS;

END_VAR

**************************************************************************
* FB EXHAUST
**************************************************************************
FUNCTION_BLOCK EXHAUST

VAR_INPUT
xEnab:          BOOL;       * =1 enabled
x5axes:         BYTE;       * =1 Gestione 5 assi
xNumXaxis:      BYTE;       * asse X
xNumYaxis:      BYTE;       * asse Y
xQtaSovrap:     DWORD;      * Quota sovrapposizione
xTimerOff:      DWORD;      * Timer off
END_VAR

VAR_OUTPUT
yOut1:          DWORD;      * Uscite
END_VAR

VAR
END_VAR
**************************************************************************

LD   xEnab                         ** =1 enabled
JMPCN ExitExhaust

LD   xQtaSovrap                    ** Quota sovrapposizione
ST   %GenVasche.GV_ParDW0

LD   xTimerOff                     ** Timer off
ST   %GenVasche.GV_ParDW1

LD   x5axes                        ** =1 Gestione 5 assi
ST   %GenVasche.GV_ParB0

LD   xNumXaxis                     ** asse X
ST   %GenVasche.GV_ParB1

LD   xNumYaxis                     ** asse Y
ST   %GenVasche.GV_ParB2

LD   %Bocca0.QStart     * Quota inizio bocca di aspirazione
ST   VASCA0.xStartX     * Quota inizio vasca (micron)
LD   %Bocca0.QEnd       * Quota fine bocca di aspirazione
ST   VASCA0.xEndX       * Quota fine vasca (micron)

LD   %Bocca0.QStartY    * Quota inizio bocca di aspirazione
ST   VASCA0.xStartY     * Quota inizio vasca (micron)
LD   %Bocca0.QEndY      * Quota fine bocca di aspirazione
ST   VASCA0.xEndY       * Quota fine vasca (micron)

CAL  VASCA0
***

LD   %Bocca1.QStart     * Quota inizio bocca di aspirazione
ST   VASCA1.xStartX     * Quota inizio vasca (micron)
LD   %Bocca1.QEnd       * Quota fine bocca di aspirazione
ST   VASCA1.xEndX       * Quota fine vasca (micron)

LD   %Bocca1.QStartY    * Quota inizio bocca di aspirazione
ST   VASCA1.xStartY     * Quota inizio vasca (micron)
LD   %Bocca1.QEndY      * Quota fine bocca di aspirazione
ST   VASCA1.xEndY       * Quota fine vasca (micron)

CAL  VASCA1
***

LD   %Bocca2.QStart     * Quota inizio bocca di aspirazione
ST   VASCA2.xStartX     * Quota inizio vasca (micron)
LD   %Bocca2.QEnd       * Quota fine bocca di aspirazione
ST   VASCA2.xEndX       * Quota fine vasca (micron)

LD   %Bocca2.QStartY    * Quota inizio bocca di aspirazione
ST   VASCA2.xStartY     * Quota inizio vasca (micron)
LD   %Bocca2.QEndY      * Quota fine bocca di aspirazione
ST   VASCA2.xEndY       * Quota fine vasca (micron)

CAL  VASCA2
***

LD   %Bocca3.QStart     * Quota inizio bocca di aspirazione
ST   VASCA3.xStartX     * Quota inizio vasca (micron)
LD   %Bocca3.QEnd       * Quota fine bocca di aspirazione
ST   VASCA3.xEndX       * Quota fine vasca (micron)

LD   %Bocca3.QStartY    * Quota inizio bocca di aspirazione
ST   VASCA3.xStartY     * Quota inizio vasca (micron)
LD   %Bocca3.QEndY      * Quota fine bocca di aspirazione
ST   VASCA3.xEndY       * Quota fine vasca (micron)

CAL  VASCA3
***

LD   %Bocca4.QStart     * Quota inizio bocca di aspirazione
ST   VASCA4.xStartX     * Quota inizio vasca (micron)
LD   %Bocca4.QEnd       * Quota fine bocca di aspirazione
ST   VASCA4.xEndX       * Quota fine vasca (micron)

LD   %Bocca4.QStartY    * Quota inizio bocca di aspirazione
ST   VASCA4.xStartY     * Quota inizio vasca (micron)
LD   %Bocca4.QEndY      * Quota fine bocca di aspirazione
ST   VASCA4.xEndY       * Quota fine vasca (micron)

CAL  VASCA4
***

LD   %Bocca5.QStart     * Quota inizio bocca di aspirazione
ST   VASCA5.xStartX     * Quota inizio vasca (micron)
LD   %Bocca5.QEnd       * Quota fine bocca di aspirazione
ST   VASCA5.xEndX       * Quota fine vasca (micron)

LD   %Bocca5.QStartY    * Quota inizio bocca di aspirazione
ST   VASCA5.xStartY     * Quota inizio vasca (micron)
LD   %Bocca5.QEndY      * Quota fine bocca di aspirazione
ST   VASCA5.xEndY       * Quota fine vasca (micron)

CAL  VASCA5
***

LD   %Bocca6.QStart     * Quota inizio bocca di aspirazione
ST   VASCA6.xStartX     * Quota inizio vasca (micron)
LD   %Bocca6.QEnd       * Quota fine bocca di aspirazione
ST   VASCA6.xEndX       * Quota fine vasca (micron)

LD   %Bocca6.QStartY    * Quota inizio bocca di aspirazione
ST   VASCA6.xStartY     * Quota inizio vasca (micron)
LD   %Bocca6.QEndY      * Quota fine bocca di aspirazione
ST   VASCA6.xEndY       * Quota fine vasca (micron)

CAL  VASCA6
***

LD   %Bocca7.QStart     * Quota inizio bocca di aspirazione
ST   VASCA7.xStartX     * Quota inizio vasca (micron)
LD   %Bocca7.QEnd       * Quota fine bocca di aspirazione
ST   VASCA7.xEndX       * Quota fine vasca (micron)

LD   %Bocca7.QStartY    * Quota inizio bocca di aspirazione
ST   VASCA7.xStartY     * Quota inizio vasca (micron)
LD   %Bocca7.QEndY      * Quota fine bocca di aspirazione
ST   VASCA7.xEndY       * Quota fine vasca (micron)

CAL  VASCA7
***

LD   %Bocca8.QStart     * Quota inizio bocca di aspirazione
ST   VASCA8.xStartX     * Quota inizio vasca (micron)
LD   %Bocca8.QEnd       * Quota fine bocca di aspirazione
ST   VASCA8.xEndX       * Quota fine vasca (micron)

LD   %Bocca8.QStartY    * Quota inizio bocca di aspirazione
ST   VASCA8.xStartY     * Quota inizio vasca (micron)
LD   %Bocca8.QEndY      * Quota fine bocca di aspirazione
ST   VASCA8.xEndY       * Quota fine vasca (micron)

CAL  VASCA8
***

LD   %Bocca9.QStart     * Quota inizio bocca di aspirazione
ST   VASCA9.xStartX     * Quota inizio vasca (micron)
LD   %Bocca9.QEnd       * Quota fine bocca di aspirazione
ST   VASCA9.xEndX       * Quota fine vasca (micron)

LD   %Bocca9.QStartY    * Quota inizio bocca di aspirazione
ST   VASCA9.xStartY     * Quota inizio vasca (micron)
LD   %Bocca9.QEndY      * Quota fine bocca di aspirazione
ST   VASCA9.xEndY       * Quota fine vasca (micron)

CAL  VASCA9
***

LD   %Bocca10.QStart    * Quota inizio bocca di aspirazione
ST   VASCA10.xStartX    * Quota inizio vasca (micron)
LD   %Bocca10.QEnd      * Quota fine bocca di aspirazione
ST   VASCA10.xEndX      * Quota fine vasca (micron)

LD   %Bocca10.QStartY   * Quota inizio bocca di aspirazione
ST   VASCA10.xStartY    * Quota inizio vasca (micron)
LD   %Bocca10.QEndY     * Quota fine bocca di aspirazione
ST   VASCA10.xEndY      * Quota fine vasca (micron)

CAL  VASCA10
***

LD   %Bocca11.QStart    * Quota inizio bocca di aspirazione
ST   VASCA11.xStartX    * Quota inizio vasca (micron)
LD   %Bocca11.QEnd      * Quota fine bocca di aspirazione
ST   VASCA11.xEndX      * Quota fine vasca (micron)

LD   %Bocca11.QStartY   * Quota inizio bocca di aspirazione
ST   VASCA11.xStartY    * Quota inizio vasca (micron)
LD   %Bocca11.QEndY     * Quota fine bocca di aspirazione
ST   VASCA11.xEndY      * Quota fine vasca (micron)

CAL  VASCA11
***

LD   %Bocca12.QStart    * Quota inizio bocca di aspirazione
ST   VASCA12.xStartX    * Quota inizio vasca (micron)
LD   %Bocca12.QEnd      * Quota fine bocca di aspirazione
ST   VASCA12.xEndX      * Quota fine vasca (micron)

LD   %Bocca12.QStartY   * Quota inizio bocca di aspirazione
ST   VASCA12.xStartY    * Quota inizio vasca (micron)
LD   %Bocca12.QEndY     * Quota fine bocca di aspirazione
ST   VASCA12.xEndY      * Quota fine vasca (micron)

CAL  VASCA12
***

LD   %Bocca13.QStart    * Quota inizio bocca di aspirazione
ST   VASCA13.xStartX    * Quota inizio vasca (micron)
LD   %Bocca13.QEnd      * Quota fine bocca di aspirazione
ST   VASCA13.xEndX      * Quota fine vasca (micron)

LD   %Bocca13.QStartY   * Quota inizio bocca di aspirazione
ST   VASCA13.xStartY    * Quota inizio vasca (micron)
LD   %Bocca13.QEndY     * Quota fine bocca di aspirazione
ST   VASCA13.xEndY      * Quota fine vasca (micron)

CAL  VASCA13
***

LD   %Bocca14.QStart    * Quota inizio bocca di aspirazione
ST   VASCA14.xStartX    * Quota inizio vasca (micron)
LD   %Bocca14.QEnd      * Quota fine bocca di aspirazione
ST   VASCA14.xEndX      * Quota fine vasca (micron)

LD   %Bocca14.QStartY   * Quota inizio bocca di aspirazione
ST   VASCA14.xStartY    * Quota inizio vasca (micron)
LD   %Bocca14.QEndY     * Quota fine bocca di aspirazione
ST   VASCA14.xEndY      * Quota fine vasca (micron)

CAL  VASCA14
***

LD   %Bocca15.QStart    * Quota inizio bocca di aspirazione
ST   VASCA15.xStartX    * Quota inizio vasca (micron)
LD   %Bocca15.QEnd      * Quota fine bocca di aspirazione
ST   VASCA15.xEndX      * Quota fine vasca (micron)

LD   %Bocca15.QStartY   * Quota inizio bocca di aspirazione
ST   VASCA15.xStartY    * Quota inizio vasca (micron)
LD   %Bocca15.QEndY     * Quota fine bocca di aspirazione
ST   VASCA15.xEndY      * Quota fine vasca (micron)

CAL  VASCA15
***

LD   %Bocca16.QStart    * Quota inizio bocca di aspirazione
ST   VASCA16.xStartX    * Quota inizio vasca (micron)
LD   %Bocca16.QEnd      * Quota fine bocca di aspirazione
ST   VASCA16.xEndX      * Quota fine vasca (micron)

LD   %Bocca16.QStartY   * Quota inizio bocca di aspirazione
ST   VASCA16.xStartY    * Quota inizio vasca (micron)
LD   %Bocca16.QEndY     * Quota fine bocca di aspirazione
ST   VASCA16.xEndY      * Quota fine vasca (micron)

CAL  VASCA16
***

LD   %Bocca17.QStart    * Quota inizio bocca di aspirazione
ST   VASCA17.xStartX    * Quota inizio vasca (micron)
LD   %Bocca17.QEnd      * Quota fine bocca di aspirazione
ST   VASCA17.xEndX      * Quota fine vasca (micron)

LD   %Bocca17.QStartY   * Quota inizio bocca di aspirazione
ST   VASCA17.xStartY    * Quota inizio vasca (micron)
LD   %Bocca17.QEndY     * Quota fine bocca di aspirazione
ST   VASCA17.xEndY      * Quota fine vasca (micron)

CAL  VASCA17
***

LD   %Bocca18.QStart    * Quota inizio bocca di aspirazione
ST   VASCA18.xStartX    * Quota inizio vasca (micron)
LD   %Bocca18.QEnd      * Quota fine bocca di aspirazione
ST   VASCA18.xEndX      * Quota fine vasca (micron)

LD   %Bocca18.QStartY   * Quota inizio bocca di aspirazione
ST   VASCA18.xStartY    * Quota inizio vasca (micron)
LD   %Bocca18.QEndY     * Quota fine bocca di aspirazione
ST   VASCA18.xEndY      * Quota fine vasca (micron)

CAL  VASCA18
***

LD   %Bocca19.QStart    * Quota inizio bocca di aspirazione
ST   VASCA19.xStartX    * Quota inizio vasca (micron)
LD   %Bocca19.QEnd      * Quota fine bocca di aspirazione
ST   VASCA19.xEndX      * Quota fine vasca (micron)

LD   %Bocca19.QStartY   * Quota inizio bocca di aspirazione
ST   VASCA19.xStartY    * Quota inizio vasca (micron)
LD   %Bocca19.QEndY     * Quota fine bocca di aspirazione
ST   VASCA19.xEndY      * Quota fine vasca (micron)

CAL  VASCA19
***

LD   %Bocca20.QStart    * Quota inizio bocca di aspirazione
ST   VASCA20.xStartX    * Quota inizio vasca (micron)
LD   %Bocca20.QEnd      * Quota fine bocca di aspirazione
ST   VASCA20.xEndX      * Quota fine vasca (micron)

LD   %Bocca20.QStartY   * Quota inizio bocca di aspirazione
ST   VASCA20.xStartY    * Quota inizio vasca (micron)
LD   %Bocca20.QEndY     * Quota fine bocca di aspirazione
ST   VASCA20.xEndY      * Quota fine vasca (micron)

CAL  VASCA20
***

LD   %Bocca21.QStart    * Quota inizio bocca di aspirazione
ST   VASCA21.xStartX    * Quota inizio vasca (micron)
LD   %Bocca21.QEnd      * Quota fine bocca di aspirazione
ST   VASCA21.xEndX      * Quota fine vasca (micron)

LD   %Bocca21.QStartY   * Quota inizio bocca di aspirazione
ST   VASCA21.xStartY    * Quota inizio vasca (micron)
LD   %Bocca21.QEndY     * Quota fine bocca di aspirazione
ST   VASCA21.xEndY      * Quota fine vasca (micron)

CAL  VASCA21
***

LD   %Bocca22.QStart    * Quota inizio bocca di aspirazione
ST   VASCA22.xStartX    * Quota inizio vasca (micron)
LD   %Bocca22.QEnd      * Quota fine bocca di aspirazione
ST   VASCA22.xEndX      * Quota fine vasca (micron)

LD   %Bocca22.QStartY   * Quota inizio bocca di aspirazione
ST   VASCA22.xStartY    * Quota inizio vasca (micron)
LD   %Bocca22.QEndY     * Quota fine bocca di aspirazione
ST   VASCA22.xEndY      * Quota fine vasca (micron)

CAL  VASCA22
***

LD   %Bocca23.QStart    * Quota inizio bocca di aspirazione
ST   VASCA23.xStartX    * Quota inizio vasca (micron)
LD   %Bocca23.QEnd      * Quota fine bocca di aspirazione
ST   VASCA23.xEndX      * Quota fine vasca (micron)

LD   %Bocca23.QStartY   * Quota inizio bocca di aspirazione
ST   VASCA23.xStartY    * Quota inizio vasca (micron)
LD   %Bocca23.QEndY     * Quota fine bocca di aspirazione
ST   VASCA23.xEndY      * Quota fine vasca (micron)

CAL  VASCA23
***

LD   %Bocca24.QStart    * Quota inizio bocca di aspirazione
ST   VASCA24.xStartX    * Quota inizio vasca (micron)
LD   %Bocca24.QEnd      * Quota fine bocca di aspirazione
ST   VASCA24.xEndX      * Quota fine vasca (micron)

LD   %Bocca24.QStartY   * Quota inizio bocca di aspirazione
ST   VASCA24.xStartY    * Quota inizio vasca (micron)
LD   %Bocca24.QEndY     * Quota fine bocca di aspirazione
ST   VASCA24.xEndY      * Quota fine vasca (micron)

CAL  VASCA24
***

LD   %Bocca25.QStart    * Quota inizio bocca di aspirazione
ST   VASCA25.xStartX    * Quota inizio vasca (micron)
LD   %Bocca25.QEnd      * Quota fine bocca di aspirazione
ST   VASCA25.xEndX      * Quota fine vasca (micron)

LD   %Bocca25.QStartY   * Quota inizio bocca di aspirazione
ST   VASCA25.xStartY    * Quota inizio vasca (micron)
LD   %Bocca25.QEndY     * Quota fine bocca di aspirazione
ST   VASCA25.xEndY      * Quota fine vasca (micron)

CAL  VASCA25
***

LD   %Bocca26.QStart    * Quota inizio bocca di aspirazione
ST   VASCA26.xStartX    * Quota inizio vasca (micron)
LD   %Bocca26.QEnd      * Quota fine bocca di aspirazione
ST   VASCA26.xEndX      * Quota fine vasca (micron)

LD   %Bocca26.QStartY   * Quota inizio bocca di aspirazione
ST   VASCA26.xStartY    * Quota inizio vasca (micron)
LD   %Bocca26.QEndY     * Quota fine bocca di aspirazione
ST   VASCA26.xEndY      * Quota fine vasca (micron)

CAL  VASCA26
***

LD   %Bocca27.QStart    * Quota inizio bocca di aspirazione
ST   VASCA27.xStartX    * Quota inizio vasca (micron)
LD   %Bocca27.QEnd      * Quota fine bocca di aspirazione
ST   VASCA27.xEndX      * Quota fine vasca (micron)

LD   %Bocca27.QStartY   * Quota inizio bocca di aspirazione
ST   VASCA27.xStartY    * Quota inizio vasca (micron)
LD   %Bocca27.QEndY     * Quota fine bocca di aspirazione
ST   VASCA27.xEndY      * Quota fine vasca (micron)

CAL  VASCA27
***

LD   %Bocca28.QStart    * Quota inizio bocca di aspirazione
ST   VASCA28.xStartX    * Quota inizio vasca (micron)
LD   %Bocca28.QEnd      * Quota fine bocca di aspirazione
ST   VASCA28.xEndX      * Quota fine vasca (micron)

LD   %Bocca28.QStartY   * Quota inizio bocca di aspirazione
ST   VASCA28.xStartY    * Quota inizio vasca (micron)
LD   %Bocca28.QEndY     * Quota fine bocca di aspirazione
ST   VASCA28.xEndY      * Quota fine vasca (micron)

CAL  VASCA28
***

LD   %Bocca29.QStart    * Quota inizio bocca di aspirazione
ST   VASCA29.xStartX    * Quota inizio vasca (micron)
LD   %Bocca29.QEnd      * Quota fine bocca di aspirazione
ST   VASCA29.xEndX      * Quota fine vasca (micron)

LD   %Bocca29.QStartY   * Quota inizio bocca di aspirazione
ST   VASCA29.xStartY    * Quota inizio vasca (micron)
LD   %Bocca29.QEndY     * Quota fine bocca di aspirazione
ST   VASCA29.xEndY      * Quota fine vasca (micron)

CAL  VASCA29
***

LD   %Bocca30.QStart    * Quota inizio bocca di aspirazione
ST   VASCA30.xStartX    * Quota inizio vasca (micron)
LD   %Bocca30.QEnd      * Quota fine bocca di aspirazione
ST   VASCA30.xEndX      * Quota fine vasca (micron)

LD   %Bocca30.QStartY   * Quota inizio bocca di aspirazione
ST   VASCA30.xStartY    * Quota inizio vasca (micron)
LD   %Bocca30.QEndY     * Quota fine bocca di aspirazione
ST   VASCA30.xEndY      * Quota fine vasca (micron)

CAL  VASCA30
***

LD   %Bocca31.QStart    * Quota inizio bocca di aspirazione
ST   VASCA31.xStartX    * Quota inizio vasca (micron)
LD   %Bocca31.QEnd      * Quota fine bocca di aspirazione
ST   VASCA31.xEndX      * Quota fine vasca (micron)

LD   %Bocca31.QStartY   * Quota inizio bocca di aspirazione
ST   VASCA31.xStartY    * Quota inizio vasca (micron)
LD   %Bocca31.QEndY     * Quota fine bocca di aspirazione
ST   VASCA31.xEndY      * Quota fine vasca (micron)

CAL  VASCA31
***

*** GESTIONE USCITE LOGICHE

LD   VASCA0.yVascaOn     * Apri vasca
ST   yOut1.0
LD   VASCA1.yVascaOn     * Apri vasca
ST   yOut1.1
LD   VASCA2.yVascaOn     * Apri vasca
ST   yOut1.2
LD   VASCA3.yVascaOn     * Apri vasca
ST   yOut1.3
LD   VASCA4.yVascaOn     * Apri vasca
ST   yOut1.4
LD   VASCA5.yVascaOn     * Apri vasca
ST   yOut1.5
LD   VASCA6.yVascaOn     * Apri vasca
ST   yOut1.6
LD   VASCA7.yVascaOn     * Apri vasca
ST   yOut1.7
LD   VASCA8.yVascaOn     * Apri vasca
ST   yOut1.8
LD   VASCA9.yVascaOn     * Apri vasca
ST   yOut1.9
LD   VASCA10.yVascaOn    * Apri vasca
ST   yOut1.10
LD   VASCA11.yVascaOn    * Apri vasca
ST   yOut1.11
LD   VASCA12.yVascaOn    * Apri vasca
ST   yOut1.12
LD   VASCA13.yVascaOn    * Apri vasca
ST   yOut1.13
LD   VASCA14.yVascaOn    * Apri vasca
ST   yOut1.14
LD   VASCA15.yVascaOn    * Apri vasca
ST   yOut1.15
LD   VASCA16.yVascaOn    * Apri vasca
ST   yOut1.16
LD   VASCA17.yVascaOn    * Apri vasca
ST   yOut1.17
LD   VASCA18.yVascaOn    * Apri vasca
ST   yOut1.18
LD   VASCA19.yVascaOn    * Apri vasca
ST   yOut1.19
LD   VASCA20.yVascaOn    * Apri vasca
ST   yOut1.20
LD   VASCA21.yVascaOn    * Apri vasca
ST   yOut1.21
LD   VASCA22.yVascaOn    * Apri vasca
ST   yOut1.22
LD   VASCA23.yVascaOn    * Apri vasca
ST   yOut1.23
LD   VASCA24.yVascaOn    * Apri vasca
ST   yOut1.24
LD   VASCA25.yVascaOn    * Apri vasca
ST   yOut1.25
LD   VASCA26.yVascaOn    * Apri vasca
ST   yOut1.26
LD   VASCA27.yVascaOn    * Apri vasca
ST   yOut1.27
LD   VASCA28.yVascaOn    * Apri vasca
ST   yOut1.28
LD   VASCA29.yVascaOn    * Apri vasca
ST   yOut1.29
LD   VASCA30.yVascaOn    * Apri vasca
ST   yOut1.30
LD   VASCA31.yVascaOn    * Apri vasca
ST   yOut1.31

ExitExhaust:

END_FUNCTION_BLOCK

(* ---- SPist.plc ---- *)
**********************************************
********** SINGLE PISTON MANAGEMENT **********
**********************************************

VAR
#include "Cnc.inc"
END_VAR

FUNCTION_BLOCK SINGLE_PISTON

VAR_INPUT
xEmerg:	                      BOOL;
xAuto:	                      BOOL;
xReset:                       BOOL;
xManualPlus:	                BOOL;
xManualMinus:                 BOOL;
xAutoPlus:                    BOOL;
xAutoMinus:                   BOOL;
xAirPressure:                 BOOL;
xSensorPlus:                  BOOL;
xSensorMinus:                 BOOL;
xSingleEffect:                BOOL;
xTimeOut:                    DWORD;
xPlusAtInit:                  BOOL;
END_VAR

VAR_OUTPUT
yPistonPlus:                  BOOL;
yPistonMinus:                 BOOL;
yWaitMFun:                    BOOL;
yAlarm:                       BOOL;      * movement commanded but not executed
yAlarm1:                      BOOL;      * movement request but not allowed
END_VAR

VAR
St_Minus:                     BOOL;
St_Plus:                      BOOL;
Ton_Minus:                     TON;
Ton_Plus:                      TON;

END_VAR

** IN STATE
LD  St_Plus
AND(
LD  xAuto
AND xAutoMinus
OR(
LDN xAuto
AND xManualMinus
)
)
OR(
LD   St_Minus
ANDN St_Plus
)
OR(
LD   ON_ONE_SCAN                   ** PLCFLAGS.8  Flag on alla prima scansione PLC
ANDN xPlusAtInit
)
ST  St_Minus

** OUT STATE
LD  St_Minus
AND(
LD  xAuto
AND xAutoPlus
OR(
LDN xAuto
AND xManualPlus
)
)
OR(
LD   St_Plus
ANDN St_Minus
)
OR(
LD   ON_ONE_SCAN                   ** PLCFLAGS.8  Flag on alla prima scansione PLC
AND  xPlusAtInit
)
ST  St_Plus

** Outputs
LD  St_Plus
*AND xEmerg
AND xAirPressure
ST  yPistonPlus

LD  St_Minus
*AND xEmerg
AND xAirPressure
ST  yPistonMinus

** Alarm
CAL Ton_Plus(IN:=yPistonPlus, PT=xTimeOut)

CAL  Ton_Minus(IN:=yPistonMinus, PT=xTimeOut)

LD   Ton_Plus.Q
ANDN xSensorPlus
OR(
LD   Ton_Minus.Q
ANDN xSensorMinus
ANDN xSingleEffect
)
S    yAlarm                        ** movement commanded but not executed

LD   xReset
R    yAlarm                        ** movement commanded but not executed

*
LD   xManualPlus
OR   xAutoPlus
ANDN xSensorPlus
OR   (
LD   xManualMinus
OR   xAutoMinus
ANDN xSensorMinus
)
ANDN xEmerg
S    yAlarm1                       ** movement request but not allowed

LD   xReset
R    yAlarm1                       ** movement request but not allowed

LD   St_Plus
ANDN xSensorPlus
OR(
LD   St_Minus
ANDN xSensorMinus
ANDN xSingleEffect
)
OR   yAlarm                        ** movement commanded but not executed
ST   yWaitMFun

END_FUNCTION_BLOCK
